FUNCTION_BLOCK T_AddCustomPackModeSetsCorrectly EXTENDS T_UnitTestBase
VAR
  mockState : T_MockStateModule;
  modeManager : T_ModeManager(mockState);

  customMode : T_BaseMode;
  expected, actual : I_PackMode;

  result : BOOL;
END_VAR

modemanager.AddCustomPackMode(0, customMode);
actual := modeManager.CustomPackModes[0];
expected := customMode;
result := actual = expected;
assertion.AssertEquals_BOOL(TRUE, result, 'result := actual = expected;');
TestFinished();

END_FUNCTION_BLOCK

(* stored: Version 1.1.0.1, ProductVersion 3.1.4024.12
   POU T_AddCustomPackModeSetsCorrectly: Id {e829e8cc-688d-4c43-b94f-41c994699b59}, SpecialFunc None *)
